TYPE T_Ctrl_SIf_IBH_Cur :
STRUCT
END_STRUCT
END_TYPE

(* stored: Version 1.1.0.1, ProductVersion 3.1.0.25
   DUT T_Ctrl_SIf_IBH_Cur: Id {491621bb-4870-4bbd-b8aa-17de8d584c9e} *)
